{attribute 'GeneratedUsingTerminal: EK1122-0000-0018'}
{attribute addProperty BoxType "EK1122-0000-0018"}
{attribute addProperty Id "RC20_VI_AES_D_BC_ECAT_xAES_A3B0707168RC20_SAFETY_Flexi_Soft_EtherCAT_GatewayFlexi_Soft_EtherCAT_Gateway_DE394EDD5"}
{attribute addProperty CRC "1999773031"}
{attribute addProperty Size "73"}
{attribute addProperty Name "RC20_A2 (EK1122)"}
TYPE RC20_A2_EK1122_77321D67 EXTENDS EK1122_1FC0878B :
STRUCT
	{attribute addProperty Name "RC20_VI (AES-D-BC-ECAT)"}
	{attribute addProperty PreviousPort "RC20_A2 (EK1122) : D"}
	RC20_VI_AES_D_BC_ECAT_x : AES_A3B07071;
	{attribute addProperty Name "RC20_SAFETY (Flexi Soft EtherCAT Gateway)"}
	{attribute addProperty PreviousPort "RC20_A2 (EK1122) : B"}
	RC20_SAFETY_Flexi_Soft_EtherCAT_Gateway : Flexi_Soft_EtherCAT_Gateway_DE394EDD;
END_STRUCT
END_TYPE

(* stored: Version 1.2.0.0, ProductVersion 3.1.4024.11
   DUT RC20_A2_EK1122_77321D67: Id {b2caec51-029a-05dd-1527-a4dc2e16774b} *)
